// ---- VISUs/Manual_Camera_RawData.TcVIS
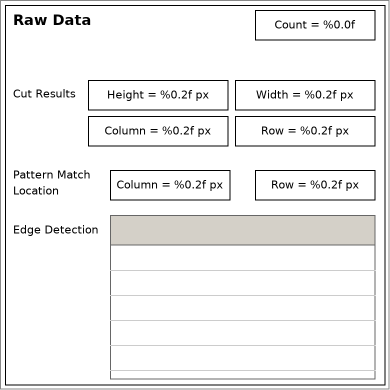
VISUALIZATION Manual_Camera_RawData  // 390x390
    Rectangle (5,5 380x380)
    Label (10,5 297x30), "Raw Data"
    Rectangle (255,10 120x30), "Count = %0.0f", text variable: MAIN.fbSlitter.Camera.CameraData.Results.Count
    Rectangle (110,170 120x30), "Column = %0.2f px", text variable: MAIN.fbSlitter.Camera.CameraData.Results.PatternMatchColumn
    Rectangle (255,170 120x30), "Row = %0.2f px", text variable: MAIN.fbSlitter.Camera.CameraData.Results.PatternMatchRow
    Rectangle (88,116 140x30), "Column = %0.2f px", text variable: MAIN.fbSlitter.Camera.CameraData.Results.LocationInX
    Rectangle (235,116 140x30), "Row = %0.2f px", text variable: MAIN.fbSlitter.Camera.CameraData.Results.LocationInY
    Rectangle (88,80 140x30), "Height = %0.2f px", text variable: MAIN.fbSlitter.Camera.CameraData.Results.HeightMeasurement
    Rectangle (235,80 140x30), "Width = %0.2f px", text variable: MAIN.fbSlitter.Camera.CameraData.Results.WidthMeasurement
    Label (10,215 101x30), "Edge Detection"
    Table (110,215 265x164), data array: MAIN.fbSlitter.Camera._displayVisionPts
        p1128707560: GVL.NumberVisionPoints
        p3854506369: MAIN.fbSlitter.Camera._displayVisionPts[1,INDEX]
        p1892666644: MAIN.fbSlitter.Camera._displayVisionPts[2,INDEX]
        p2232123230: Column
        p511219082: Row
    Group (10,160 96x46)
        Label (0,0 96x30), "Pattern Match"
        Label (0,16 96x30), "Location"
    Label (10,79 101x30), "Cut Results"
END_VISUALIZATION

// ---- VISUs/Manual_Cutter.TcVIS
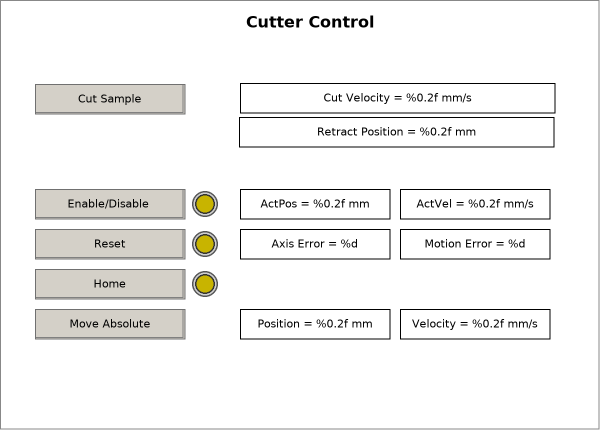
VISUALIZATION Manual_Cutter  // 600x430
    Label (133,7 355x30), "Cutter Control"
    Button (35,84 150x30), "Cut Sample", input disabled if: MAIN.fbSlitter.bBusy
        OnMouseClick: execute { MAIN.fbSlitter.Manual.bCutSample := TRUE; }
    Button (35,189 150x30), "Enable/Disable", input disabled if: MAIN.fbSlitter.bBusy
        OnMouseClick: execute { MAIN.fbSlitter.Manual.bCutterDisable := TRUE; }
    Button (35,229 150x30), "Reset", input disabled if: MAIN.fbSlitter.bBusy
        OnMouseClick: execute { MAIN.fbSlitter.Manual.bCutterReset := TRUE; }
    Button (35,269 150x30), "Home"
        OnMouseClick: execute { MAIN.fbSlitter.Manual.bCutterHome := TRUE; }
    Lamp1 (190,189 30x30), variable: MAIN.fbSlitter.Cutter.Axis.NcToPlc.StateDWord.0 = 1, style: Lamp-Lamp1-Yellow
    Rectangle (240,229 150x30), "Axis Error = %d", text variable: MAIN.fbSlitter.Cutter.Axis.NcToPlc.ErrorCode
    Lamp1 (190,229 30x30), variable: MAIN.fbSlitter.Cutter.Axis.NcToPlc.ErrorCode <> 0, style: Lamp-Lamp1-Yellow
    Lamp1 (190,269 30x30), variable: MAIN.fbSlitter.Cutter.Axis.NcToPlc.StateDWord.1 = 1, style: Lamp-Lamp1-Yellow
    Rectangle (400,229 150x30), "Motion Error = %d", text variable: MAIN.fbSlitter.Cutter._errorCode
    Button (35,309 150x30), "Move Absolute"
        OnMouseClick: execute { MAIN.fbSlitter.Manual.bCutterMoveAbs := TRUE; }
    Rectangle (240,309 150x30), "Position = %0.2f mm", text variable: MAIN.fbSlitter.Cutter._position
        OnMouseClick: write MAIN.fbSlitter.Cutter._position via Default, min 0, max 20, title 'Cutter Position'
    Rectangle (400,309 150x30), "Velocity = %0.2f mm/s", text variable: MAIN.fbSlitter.Cutter._velocity
        OnMouseClick: write MAIN.fbSlitter.Cutter._velocity via Default, title 'Cutter Velocity'
    Rectangle (240,189 150x30), "ActPos = %0.2f mm", text variable: MAIN.fbSlitter.Cutter.Axis.NcToPlc.ActPos
    Rectangle (400,189 150x30), "ActVel = %0.2f mm/s", text variable: MAIN.fbSlitter.Cutter.Axis.NcToPlc.ActVelo
    Rectangle (240,83 315x30), "Cut Velocity = %0.2f mm/s", text variable: MAIN.fbSlitter.Cutter._hmiParameters.cutVelocity
        OnMouseClick: write MAIN.fbSlitter.Cutter._hmiParameters.cutVelocity via Default, title 'Cutter Velocity'
    Rectangle (239,117 315x30), "Retract Position = %0.2f mm", text variable: MAIN.fbSlitter.Cutter._hmiParameters.retractPosition
        OnMouseClick: write MAIN.fbSlitter.Cutter._hmiParameters.retractPosition via Default, title 'Retract Position'
END_VISUALIZATION

// ---- VISUs/Manual_Ejector.TcVIS
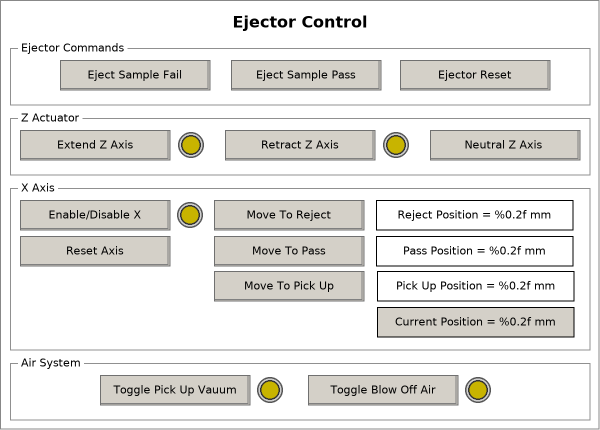
VISUALIZATION Manual_Ejector  // 600x430
    GroupBox (10,355 580x65), "Air System"
    Label (0,7 600x30), "Ejector Control"
    Button (100,375 150x30), "Toggle Pick Up Vauum"
        OnMouseClick: execute { MAIN.fbSlitter.Manual.bEjectVacuum := TRUE; }
    Button (308,375 150x30), "Toggle Blow Off Air"
        OnMouseClick: execute { MAIN.fbSlitter.Manual.bEjectBlowOff := TRUE; }
    Lamp1 (463,375 30x30), variable: MAIN.fbSlitter.Ejector._BlowOff, style: Lamp-Lamp1-Yellow
    Lamp1 (255,375 30x30), variable: MAIN.fbSlitter.Ejector._Vacuum, style: Lamp-Lamp1-Yellow
    Group (10,110 580x65)
        GroupBox (0,0 580x65), "Z Actuator"
        Button (10,20 150x30), "Extend Z Axis", input disabled if: MAIN.fbSlitter.bBusy
            OnMouseClick: execute { MAIN.fbSlitter.Manual.bEjectZExtend := TRUE; }
        Button (215,20 150x30), "Retract Z Axis", input disabled if: MAIN.fbSlitter.bBusy
            OnMouseClick: execute { MAIN.fbSlitter.Manual.bEjectZRetract := TRUE; }
        Button (420,20 150x30), "Neutral Z Axis", input disabled if: MAIN.fbSlitter.bBusy
            tap MAIN.fbSlitter.Manual.bEjectZOff
            OnMouseClick: execute { MAIN.fbSlitter.Manual.bEjectZNeutral := TRUE; }
        Lamp1 (166,20 30x30), variable: MAIN.fbSlitter.Ejector.zSlide.diExtended, style: Lamp-Lamp1-Yellow
        Lamp1 (371,20 30x30), variable: MAIN.fbSlitter.Ejector.zSlide.diRetracted, style: Lamp-Lamp1-Yellow
    GroupBox (10,40 580x65), "Ejector Commands"
        Button (390,20 150x30), "Ejector Reset", input disabled if: MAIN.fbSlitter.bBusy
            OnMouseClick: execute { MAIN.fbSlitter.Manual.bEjectReset := TRUE; }
    Button (60,60 150x30), "Eject Sample Fail", input disabled if: MAIN.fbSlitter.bBusy
        OnMouseClick: execute { MAIN.fbSlitter.Manual.bEjectSampleFail := TRUE; }
    Button (231,60 150x30), "Eject Sample Pass", input disabled if: MAIN.fbSlitter.bBusy
        OnMouseClick: execute { MAIN.fbSlitter.Manual.bEjectSamplePass := TRUE; }
    GroupBox (10,180 580x170), "X Axis"
        Rectangle (367,91 197x30), "Pick Up Position = %0.2f mm", text variable: MAIN.fbSlitter.Ejector._hmiParameters.ejectPositionHome
            OnMouseClick: write MAIN.fbSlitter.Ejector._hmiParameters.ejectPositionHome via Default, title 'Pick Up Position'
        Rectangle (367,127 197x30), "Current Position = %0.2f mm", text variable: MAIN.fbSlitter.Ejector.axis.axis.NcToPlc.ActPos
        Button (10,56 150x30), "Reset Axis"
            OnMouseClick: execute { MAIN.fbSlitter.Manual.bEjectAxisReset := TRUE; }
    Button (20,200 150x30), "Enable/Disable X", input disabled if: MAIN.fbSlitter.bBusy
        OnMouseClick: execute { MAIN.fbSlitter.Manual.bEjectAxisEnableToggle := TRUE; }
    Lamp1 (175,200 30x30), variable: MAIN.fbSlitter.Ejector.axis.axis.NcToPlc.StateDWord.0 = 1, style: Lamp-Lamp1-Yellow
    Button (214,200 150x30), "Move To Reject", input disabled if: MAIN.fbSlitter.bBusy
        OnMouseClick: execute { Main.fbSlitter.Manual.bEjectAxisFailPosition := TRUE; }
    Button (214,236 150x30), "Move To Pass", input disabled if: MAIN.fbSlitter.bBusy
        OnMouseClick: execute { Main.fbSlitter.Manual.bEjectAxisPassPosition := TRUE; }
    Button (214,271 150x30), "Move To Pick Up", input disabled if: MAIN.fbSlitter.bBusy
        OnMouseClick: execute { Main.fbSlitter.Manual.bEjectAxisHomePosition := TRUE; }
    Rectangle (376,200 197x30), "Reject Position = %0.2f mm", text variable: MAIN.fbSlitter.Ejector._hmiParameters.ejectPositionFail
        OnMouseClick: write MAIN.fbSlitter.Ejector._hmiParameters.ejectPositionFail via Default, title 'Reject Position'
    Rectangle (376,236 197x30), "Pass Position = %0.2f mm", text variable: MAIN.fbSlitter.Ejector._hmiParameters.ejectPositionPass
        OnMouseClick: write MAIN.fbSlitter.Ejector._hmiParameters.ejectPositionPass via Default, title 'Pass Position'
END_VISUALIZATION

// ---- VISUs/Manual_Frame.TcVIS
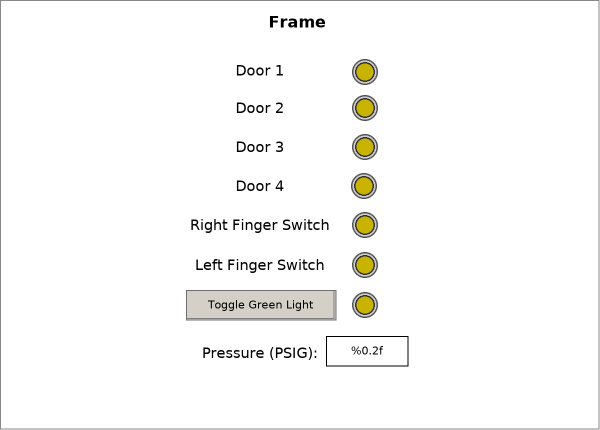
VISUALIZATION Manual_Frame  // 600x430
    Label (0,7 600x30), "Frame"
    Label (185,57 150x27), "Door 1"
    Label (185,93 150x30), "Door 2"
    Label (185,132 150x30), "Door 3"
    Label (185,210 150x30), "Right Finger Switch"
    Label (185,250 150x30), "Left Finger Switch"
    Lamp1 (350,57 30x30), variable: MAIN.Frame.diDoor1, style: Lamp-Lamp1-Yellow
    Lamp1 (350,93 30x30), variable: MAIN.Frame.diDoor2, style: Lamp-Lamp1-Yellow
    Lamp1 (350,132 30x30), variable: MAIN.Frame.diDoor3, style: Lamp-Lamp1-Yellow
    Lamp1 (350,210 30x30), variable: MAIN.Frame.diControlLeft, style: Lamp-Lamp1-Yellow
    Lamp1 (350,250 30x30), variable: MAIN.Frame.diControlRight, style: Lamp-Lamp1-Yellow
    Lamp1 (350,290 30x30), variable: MAIN.Frame.doGreen, style: Lamp-Lamp1-Yellow
    Button (186,290 150x30), "Toggle Green Light"
        OnMouseClick: execute { MAIN.Frame.GreenLight := NOT MAIN.Frame.GreenLight; }
    Label (185,338 150x30), "Pressure (PSIG):"
    Rectangle (326,336 82x30), "%0.2f", text variable: MAIN.Frame._pressure
    Label (185,171 150x30), "Door 4"
    Lamp1 (349,171 30x30), variable: MAIN.Frame.diDoor4, style: Lamp-Lamp1-Yellow
END_VISUALIZATION

// ---- VISUs/Manual_Mandrel.TcVIS
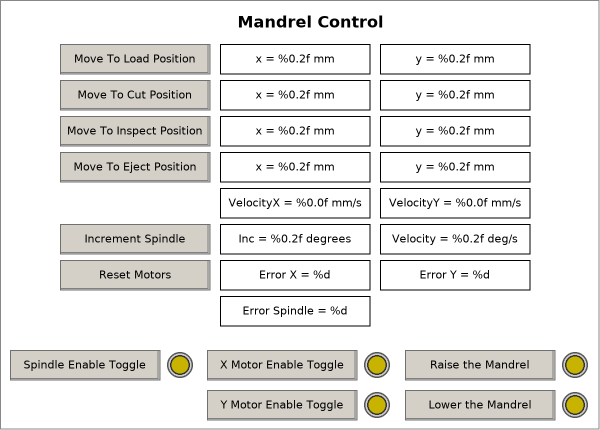
VISUALIZATION Manual_Mandrel  // 600x430
    Button (60,44 150x30), "Move To Load Position", input disabled if: MAIN.fbSlitter.bBusy
        OnMouseClick: execute { MAIN.fbSlitter.Manual.bMoveToLoadPosition := TRUE; }
    Button (60,80 150x30), "Move To Cut Position", input disabled if: MAIN.fbSlitter.bBusy
        OnMouseClick: execute { MAIN.fbSlitter.Manual.bMoveToCutPosition := TRUE; }
    Button (60,116 150x30), "Move To Inspect Position", input disabled if: MAIN.fbSlitter.bBusy
        OnMouseClick: execute { MAIN.fbSlitter.Manual.bMoveToInspectPosition := TRUE; }
    Button (60,152 150x30), "Move To Eject Position", input disabled if: MAIN.fbSlitter.bBusy
        OnMouseClick: execute { MAIN.fbSlitter.Manual.bMoveToEjectPosition := TRUE; }
    Button (405,350 150x30), "Raise the Mandrel", input disabled if: MAIN.fbSlitter.bBusy
        OnMouseClick: execute { MAIN.fbSlitter.Manual.bRaiseMandrel := TRUE; }
    Button (405,390 150x30), "Lower the Mandrel", input disabled if: MAIN.fbSlitter.bBusy
        OnMouseClick: execute { MAIN.fbSlitter.Manual.bLowerMandrel := TRUE; }
    Rectangle (220,44 150x30), "x = %0.2f mm", text variable: MAIN.fbSlitter.Mandrel._hmiParameters.loadPositionX
        OnMouseClick: write MAIN.fbSlitter.Mandrel._hmiParameters.loadPositionX via Default, title 'Load Position X'
    Rectangle (380,44 150x30), "y = %0.2f mm", text variable: MAIN.fbSlitter.Mandrel._hmiParameters.loadPositionY
        OnMouseClick: write MAIN.fbSlitter.Mandrel._hmiParameters.loadPositionY via Default, title 'Load Position Y'
    Rectangle (220,80 150x30), "x = %0.2f mm", text variable: MAIN.TubeHmi.CutPositionX
        OnMouseClick: write MAIN.TubeHmi.CutPositionX via Default, title 'Cut Position X'
    Rectangle (380,80 150x30), "y = %0.2f mm", text variable: MAIN.TubeHmi.CutPositionY
        OnMouseClick: write MAIN.TubeHmi.CutPositionY via Default, title 'Cut Position Y'
    Rectangle (220,116 150x30), "x = %0.2f mm", text variable: MAIN.TubeHmi.InspectPositionX
        OnMouseClick: write MAIN.TubeHmi.InspectPositionX via Default, title 'Inspect Position X'
    Rectangle (380,116 150x30), "y = %0.2f mm", text variable: MAIN.TubeHmi.InspectPositionY
        OnMouseClick: write MAIN.TubeHmi.InspectPositionY via Default, title 'Inspect Position Y'
    Rectangle (220,152 150x30), "x = %0.2f mm", text variable: MAIN.TubeHmi.EjectPositionX
        OnMouseClick: write MAIN.TubeHmi.EjectPositionX via Default, title 'Eject Position X'
    Rectangle (380,152 150x30), "y = %0.2f mm", text variable: MAIN.TubeHmi.EjectPositionY
        OnMouseClick: write MAIN.TubeHmi.EjectPositionY via Default, title 'Eject Position Y'
    Lamp1 (560,350 30x30), variable: MAIN.fbSlitter.Mandrel.doStripperExtend AND NOT MAIN.fbSlitter.Mandrel.doStripperRetract, style: Lamp-Lamp1-Yellow
    Lamp1 (560,390 30x30), variable: NOT MAIN.fbSlitter.Mandrel.doStripperExtend AND MAIN.fbSlitter.Mandrel.doStripperRetract, style: Lamp-Lamp1-Yellow
    Rectangle (220,188 150x30), "VelocityX = %0.0f mm/s", text variable: MAIN.fbSlitter.Mandrel._hmiParameters.velocityX
        OnMouseClick: write MAIN.fbSlitter.Mandrel._hmiParameters.velocityX via Default, title 'Velocity X'
    Rectangle (380,188 150x30), "VelocityY = %0.0f mm/s", text variable: MAIN.fbSlitter.Mandrel._hmiParameters.velocityY
        OnMouseClick: write MAIN.fbSlitter.Mandrel._hmiParameters.velocityY via Default, title 'Velocity Y'
    Rectangle (220,260 150x30), "Error X = %d", text variable: MAIN.fbSlitter.Mandrel.Xaxis.NcToPlc.ErrorCode
    Rectangle (380,260 150x30), "Error Y = %d", text variable: MAIN.fbSlitter.Mandrel.Yaxis.NcToPlc.ErrorCode
    Button (60,260 150x30), "Reset Motors"
        OnMouseClick: execute { MAIN.fbSlitter.Manual.bMandrelReset := TRUE; }
    Button (207,350 150x30), "X Motor Enable Toggle", input disabled if: MAIN.fbSlitter.bBusy
        OnMouseClick: execute { MAIN.fbSlitter.Manual.bMandrelXEnableToggle := TRUE; }
    Button (207,390 150x30), "Y Motor Enable Toggle", input disabled if: MAIN.fbSlitter.bBusy
        OnMouseClick: execute { MAIN.fbSlitter.Manual.bMandrelYEnableToggle := TRUE; }
    Button (10,350 150x30), "Spindle Enable Toggle"
        OnMouseClick: execute { MAIN.fbSlitter.Manual.bMandrelSpindleToggle := TRUE; }
    Lamp1 (362,350 30x30), variable: MAIN.fbSlitter.Mandrel.Xaxis.NcToPlc.StateDWord.0 = 1, style: Lamp-Lamp1-Yellow
    Lamp1 (165,350 30x30), variable: MAIN.fbSlitter.Mandrel.Spindle.NcToPlc.StateDWord.0 = 1, style: Lamp-Lamp1-Yellow
    Lamp1 (362,390 30x30), variable: MAIN.fbSlitter.Mandrel.Yaxis.NcToPlc.StateDWord.0 = 1, style: Lamp-Lamp1-Yellow
    Label (133,7 355x30), "Mandrel Control"
    Rectangle (220,296 150x30), "Error Spindle = %d", text variable: MAIN.fbSlitter.Mandrel.Spindle.NcToPlc.ErrorCode
    Button (60,224 150x30), "Increment Spindle", input disabled if: MAIN.fbSlitter.bBusy
        OnMouseClick: execute { MAIN.fbSlitter.Manual.bMandrelSpindleRotate := TRUE; }
    Rectangle (220,224 150x30), "Inc = %0.2f degrees", text variable: MAIN.fbSlitter.Mandrel._SpindleIncrement
        OnMouseClick: write MAIN.fbSlitter.Mandrel._SpindleIncrement via Default, title 'Spingle Increment'
    Rectangle (380,224 150x30), "Velocity = %0.2f deg/s", text variable: MAIN.fbSlitter.Mandrel._hmiParameters.spindleVelocity
        OnMouseClick: write MAIN.fbSlitter.Mandrel._hmiParameters.spindleVelocity via Default, title 'Spindle Velocity'
END_VISUALIZATION

// ---- VISUs/Manual_Vacuum.TcVIS
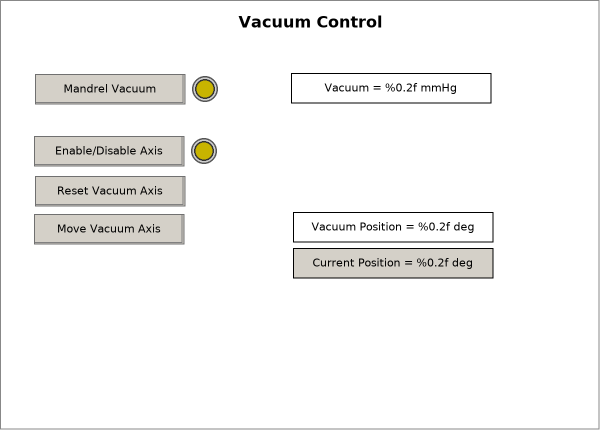
VISUALIZATION Manual_Vacuum  // 600x430
    Label (133,7 355x30), "Vacuum Control"
    Rectangle (291,73 200x30), "Vacuum = %0.2f mmHg", text variable: MAIN.fbSlitter.Mandrel._vacuum_mmHg
    Button (35,74 150x30), "Mandrel Vacuum"
        OnMouseClick: execute { MAIN.fbSlitter.Manual.bToggleMandrelVacuum := TRUE; }
    Lamp1 (190,74 30x30), variable: MAIN.fbSlitter.Mandrel.doVacuum, style: Lamp-Lamp1-Yellow
    Button (34,136 150x30), "Enable/Disable Axis"
        OnMouseClick: execute { MAIN.fbSlitter.Manual.bVacuumAxisToggleEnable := TRUE; }
    Lamp1 (189,136 30x30), variable: MAIN.fbSlitter.Mandrel.VacAxis.axis.NcToPlc.StateDWord.0 = 1, style: Lamp-Lamp1-Yellow
    Rectangle (293,248 200x30), "Current Position = %0.2f deg", text variable: MAIN.fbSlitter.Mandrel.VacAxis.axis.NcToPlc.ActPos
    Rectangle (293,212 200x30), "Vacuum Position = %0.2f deg", text variable: MAIN.TubeHmi.VacPosition
        OnMouseClick: write MAIN.TubeHmi.VacPosition via Default, min 0, max 13000, title 'Vacuum Position'
    Button (34,214 150x30), "Move Vacuum Axis"
        OnMouseClick: execute { MAIN.fbSlitter.Manual.bVacuumAxisMove := TRUE; }
    Button (35,176 150x30), "Reset Vacuum Axis"
        OnMouseClick: execute { MAIN.fbSlitter.Manual.bVacuumAxisReset := TRUE; }
END_VISUALIZATION

// ---- VISUs/Manual_Select_Tube.TcVIS
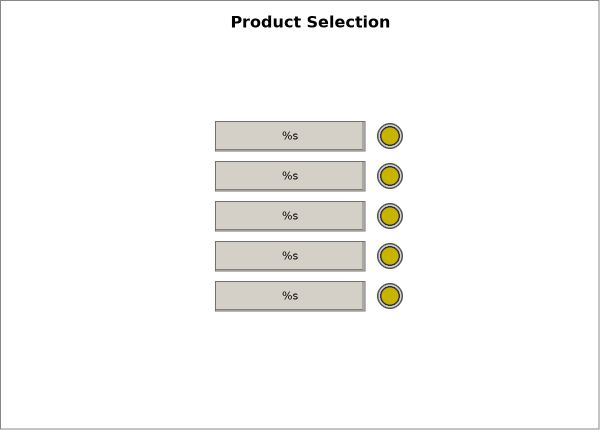
VISUALIZATION Manual_Select_Tube  // 600x430
    Button (215,121 150x30), "%s", text variable: MAIN.TubeSelection[1].ProductName
        OnMouseClick: execute {
            MAIN.TubeHmi := MAIN.TubeSelection[1];
            MAIN.fbSlitter.Manual.bCameraSelectTube := TRUE;
            MAIN.TubeIndicator[1] := TRUE;
            MAIN.TubeIndicator[2] := FALSE;
            MAIN.TubeIndicator[3] := FALSE;
            MAIN.TubeIndicator[4] := FALSE;
            MAIN.TubeIndicator[5] := FALSE;
        }
    Button (215,161 150x30), "%s", text variable: MAIN.TubeSelection[2].ProductName
        OnMouseClick: execute {
            MAIN.TubeHmi := MAIN.TubeSelection[2];
            MAIN.fbSlitter.Manual.bCameraSelectTube := TRUE;
            MAIN.TubeIndicator[1] := FALSE;
            MAIN.TubeIndicator[2] := TRUE;
            MAIN.TubeIndicator[3] := FALSE;
            MAIN.TubeIndicator[4] := FALSE;
            MAIN.TubeIndicator[5] := FALSE;
        }
    Button (215,201 150x30), "%s", text variable: MAIN.TubeSelection[3].ProductName
        OnMouseClick: execute {
            MAIN.TubeHmi := MAIN.TubeSelection[3];
            MAIN.fbSlitter.Manual.bCameraSelectTube := TRUE;
            MAIN.TubeIndicator[1] := FALSE;
            MAIN.TubeIndicator[2] := FALSE;
            MAIN.TubeIndicator[3] := TRUE;
            MAIN.TubeIndicator[4] := FALSE;
            MAIN.TubeIndicator[5] := FALSE;
        }
    Button (215,241 150x30), "%s", text variable: MAIN.TubeSelection[4].ProductName
        OnMouseClick: execute {
            MAIN.TubeHmi := MAIN.TubeSelection[4];
            MAIN.fbSlitter.Manual.bCameraSelectTube := TRUE;
            MAIN.TubeIndicator[1] := FALSE;
            MAIN.TubeIndicator[2] := FALSE;
            MAIN.TubeIndicator[3] := FALSE;
            MAIN.TubeIndicator[4] := TRUE;
            MAIN.TubeIndicator[5] := FALSE;
        }
    Button (215,281 150x30), "%s", text variable: MAIN.TubeSelection[5].ProductName
        OnMouseClick: execute {
            MAIN.TubeHmi := MAIN.TubeSelection[5];
            MAIN.fbSlitter.Manual.bCameraSelectTube := TRUE;
            MAIN.TubeIndicator[1] := FALSE;
            MAIN.TubeIndicator[2] := FALSE;
            MAIN.TubeIndicator[3] := FALSE;
            MAIN.TubeIndicator[4] := FALSE;
            MAIN.TubeIndicator[5] := TRUE;
        }
    Lamp1 (375,121 30x30), variable: MAIN.TubeIndicator[1], style: Lamp-Lamp1-Yellow
    Lamp1 (375,161 30x30), variable: MAIN.TubeIndicator[2], style: Lamp-Lamp1-Yellow
    Lamp1 (375,201 30x30), variable: MAIN.TubeIndicator[3], style: Lamp-Lamp1-Yellow
    Lamp1 (375,241 30x30), variable: MAIN.TubeIndicator[4], style: Lamp-Lamp1-Yellow
    Lamp1 (375,281 30x30), variable: MAIN.TubeIndicator[5], style: Lamp-Lamp1-Yellow
    Label (133,7 355x30), "Product Selection"
END_VISUALIZATION

// ---- VISUs/Settings.TcVIS
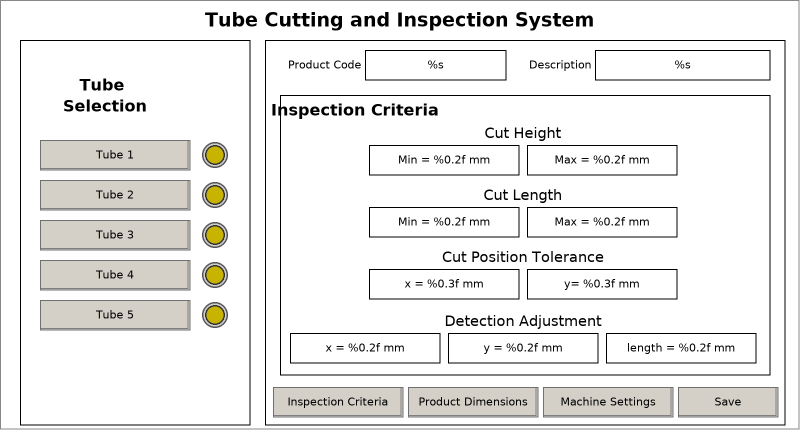
VISUALIZATION Settings  // 800x430
    Frame (255,30 540x400)
        shows SettingsTemplate(Tube := MAIN.TubeHmi)
        shows SettingsTemplate(Tube := MAIN.TubeSelection[2])
        shows SettingsTemplate(Tube := MAIN.TubeSelection[3])
        shows SettingsTemplate(Tube := MAIN.TubeSelection[4])
        shows SettingsTemplate(Tube := MAIN.TubeSelection[5])
    Label (10,79 170x30)
    Label (0,5 800x30), "Tube Cutting and Inspection System"
    Group (20,65 230x51)
        Label (0,21 170x30), "Selection"
        Label (0,0 170x30), "Tube"
    Rectangle (20,40 230x385)
    Button (40,140 150x30), "Tube 1"
        OnMouseClick: execute {
            MAIN.TubeHmi := MAIN.TubeSelection[1];
            MAIN.TubeIndicator[1] := TRUE;
            MAIN.TubeIndicator[2] := FALSE;
            MAIN.TubeIndicator[3] := FALSE;
            MAIN.TubeIndicator[4] := FALSE;
            MAIN.TubeIndicator[5] := FALSE;
        }
    Button (40,180 150x30), "Tube 2"
        OnMouseClick: execute {
            MAIN.TubeHmi := MAIN.TubeSelection[2];
            MAIN.TubeIndicator[1] := FALSE;
            MAIN.TubeIndicator[2] := TRUE;
            MAIN.TubeIndicator[3] := FALSE;
            MAIN.TubeIndicator[4] := FALSE;
            MAIN.TubeIndicator[5] := FALSE;
        }
    Button (40,220 150x30), "Tube 3"
        OnMouseClick: execute {
            MAIN.TubeHmi := MAIN.TubeSelection[3];
            MAIN.TubeIndicator[1] := FALSE;
            MAIN.TubeIndicator[2] := FALSE;
            MAIN.TubeIndicator[3] := TRUE;
            MAIN.TubeIndicator[4] := FALSE;
            MAIN.TubeIndicator[5] := FALSE;
        }
    Button (40,260 150x30), "Tube 4"
        OnMouseClick: execute {
            Main.TubeHmi := MAIN.TubeSelection[4];
            MAIN.TubeIndicator[1] := FALSE;
            MAIN.TubeIndicator[2] := FALSE;
            MAIN.TubeIndicator[3] := FALSE;
            MAIN.TubeIndicator[4] := TRUE;
            MAIN.TubeIndicator[5] := FALSE;
        }
    Button (40,300 150x30), "Tube 5"
        OnMouseClick: execute {
            Main.TubeHmi := MAIN.TubeSelection[5];
            MAIN.TubeIndicator[1] := FALSE;
            MAIN.TubeIndicator[2] := FALSE;
            MAIN.TubeIndicator[3] := FALSE;
            MAIN.TubeIndicator[4] := FALSE;
            MAIN.TubeIndicator[5] := TRUE;
        }
    Lamp1 (200,140 30x30), variable: MAIN.TubeIndicator[1], style: Lamp-Lamp1-Yellow
    Lamp1 (200,180 30x30), variable: MAIN.TubeIndicator[2], style: Lamp-Lamp1-Yellow
    Lamp1 (200,220 30x30), variable: MAIN.TubeIndicator[3], style: Lamp-Lamp1-Yellow
    Lamp1 (200,260 30x30), variable: MAIN.TubeIndicator[4], style: Lamp-Lamp1-Yellow
    Lamp1 (200,300 30x30), variable: MAIN.TubeIndicator[5], style: Lamp-Lamp1-Yellow
    Group (20,70 230x51)
        Label (0,21 170x30), "Selection"
        Label (0,0 170x30), "Tube"
END_VISUALIZATION

// ---- VISUs/SettingsTemplate.TcVIS
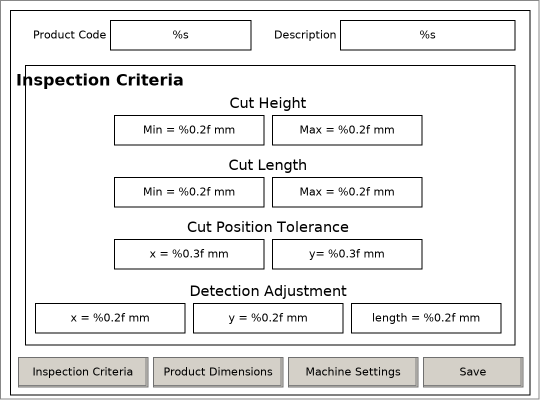
VISUALIZATION SettingsTemplate  // 540x400
VAR_IN_OUT
	Tube : ST_TubeParameters;
END_VAR
    Rectangle (10,10 520x385)
    Rectangle (110,20 141x30), "%s", text variable: Tube.ProductName
        OnMouseClick: write Tube.ProductName via Default
    Label (30,20 80x30), "Product Code"
    Button (288,357 130x30), "Machine Settings"
        OnMouseClick: FrameSelectionChange Selection=SelectedFrame=c09837a4-7cd0-42f3-a923-2461df8b3e92, Selection=1, GlobSel=AssignType=Directly, SelType=Locally
    Button (18,357 130x30), "Inspection Criteria"
        OnMouseClick: FrameSelectionChange Selection=SelectedFrame=c09837a4-7cd0-42f3-a923-2461df8b3e92, GlobSel=AssignType=Directly, SelType=Locally
    Button (153,357 130x30), "Product Dimensions"
        OnMouseClick: FrameSelectionChange Selection=SelectedFrame=c09837a4-7cd0-42f3-a923-2461df8b3e92, Selection=2, GlobSel=AssignType=Directly, SelType=Locally
    Button (423,357 100x30), "Save"
        OnMouseClick: execute { MAIN.bSave := TRUE; }
    Frame (15,55 510x300)
        shows Settings_PassCriteria(CutHeightMin := Tube.MinHeight, CutHeightMax := Tube.MaxHeight, CutLengthMin := Tube.MinLength, CutLengthMax := Tube.MaxLength, CutToleranceX := Tube.ResultToleranceX, CutToleranceY := Tube.ResultToleranceY, AdjustmentX := Tube.AdjustmentX, AdjustmentY := Tube.AdjustmentY, AdjustmentLength := Tube.AdjustmentLength)
        shows Settings_Mandrel(CutPositionX := Tube.CutPositionX, CutPositionY := Tube.CutPositionY, InspectPositionX := Tube.InspectPositionX, InspectPositionY := Tube.InspectPositionY, EjectPositionX := Tube.EjectPositionX, EjectPositionY := Tube.EjectPositionY, VacuumThreshold := Tube.VacuumThreshold, VacuumPosition := Tube.VacPosition)
        shows Settings_ProductDimensions(Diameter := Tube.Diameter, PocketDepth := Tube.DepthOfPocket)
    Label (271,20 69x30), "Description"
    Rectangle (340,20 175x30), "%s", text variable: Tube.Description
        OnMouseClick: write Tube.Description via Default
END_VISUALIZATION

// ---- VISUs/Settings_Mandrel.TcVIS
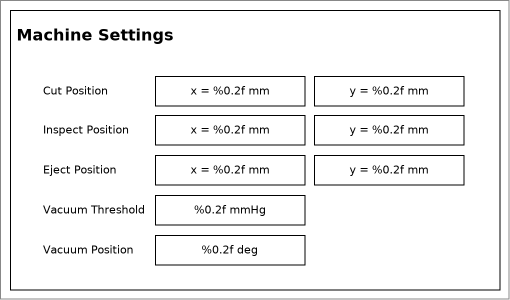
VISUALIZATION Settings_Mandrel  // 510x300
VAR_IN_OUT
	CutPositionX	: LREAL;
	CutPositionY	: LREAL;
	InspectPositionX: LREAL;
	InspectPositionY: LREAL;
	EjectPositionX	: LREAL;
	EjectPositionY	: LREAL;
	VacuumThreshold	: REAL;
	VacuumPosition : LREAL;
END_VAR
    Rectangle (10,10 490x280)
    Label (20,20 150x30), "Machine Settings"
    Label (40,76 90x30), "Cut Position"
    Label (40,115 90x30), "Inspect Position"
    Label (40,155 90x30), "Eject Position"
    Rectangle (155,76 150x30), "x = %0.2f mm", text variable: CutPositionX
        OnMouseClick: write CutPositionX via Default
    Rectangle (314,76 150x30), "y = %0.2f mm", text variable: CutPositionY
        OnMouseClick: write CutPositionY via Default
    Rectangle (155,115 150x30), "x = %0.2f mm", text variable: InspectPositionX
        OnMouseClick: write InspectPositionX via Default
    Rectangle (314,115 150x30), "y = %0.2f mm", text variable: InspectPositionY
        OnMouseClick: write InspectPositionY via Default
    Rectangle (155,155 150x30), "x = %0.2f mm", text variable: EjectPositionX
        OnMouseClick: write EjectPositionX via Default
    Rectangle (314,155 150x30), "y = %0.2f mm", text variable: EjectPositionY
        OnMouseClick: write EjectPositionY via Default
    Label (40,195 110x30), "Vacuum Threshold"
    Rectangle (155,195 150x30), "%0.2f mmHg", text variable: VacuumThreshold
        OnMouseClick: write VacuumThreshold via Default
    Label (40,235 110x30), "Vacuum Position"
    Rectangle (155,235 150x30), "%0.2f deg", text variable: VacuumPosition
        OnMouseClick: write VacuumPosition via Default, min 0, max 13000, title 'Vacuum Axis Position'
END_VISUALIZATION

// ---- VISUs/Settings_PassCriteria.TcVIS
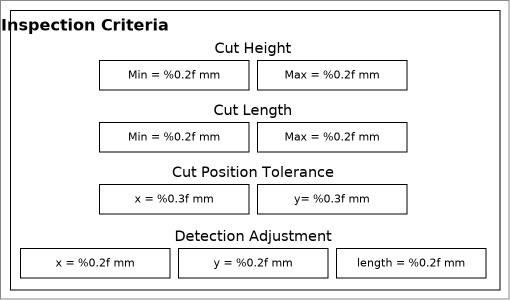
VISUALIZATION Settings_PassCriteria  // 510x300
VAR_IN_OUT
	CutHeightMin	: LREAL;
	CutHeightMax	: LREAL;
	CutLengthMin	: LREAL;
	CutLengthMax	: LREAL;
	CutToleranceX	: LREAL;
	CutToleranceY	: LREAL;
	AdjustmentX		: LREAL;
	AdjustmentY		: LREAL;
	AdjustmentLength: LREAL;
END_VAR
    Rectangle (10,10 490x280)
    Label (203,95 100x30), "Cut Length"
    Rectangle (99,122 150x30), "Min = %0.2f mm", text variable: CutLengthMin
        OnMouseClick: write CutLengthMin via Default
    Rectangle (257,122 150x30), "Max = %0.2f mm", text variable: CutLengthMax
        OnMouseClick: write CutLengthMax via Default, title 'Cut Position Y'
    Label (213,33 80x30), "Cut Height"
    Rectangle (99,60 150x30), "Min = %0.2f mm", text variable: CutHeightMin
        OnMouseClick: write CutHeightMin via Default
    Rectangle (257,60 150x30), "Max = %0.2f mm", text variable: CutHeightMax
        OnMouseClick: write CutHeightMax via Default, title 'Cut Position Y'
    Label (168,157 170x30), "Cut Position Tolerance"
    Rectangle (99,184 150x30), "x = %0.3f mm", text variable: CutToleranceX
        OnMouseClick: write CutToleranceX via Default
    Rectangle (257,184 150x30), "y= %0.3f mm", text variable: CutToleranceY
        OnMouseClick: write CutToleranceY via Default, title 'Cut Position Y'
    Label (173,221 160x30), "Detection Adjustment"
    Rectangle (20,248 150x30), "x = %0.2f mm", text variable: AdjustmentX
        OnMouseClick: write AdjustmentX via Default, title 'Cut Position X'
    Rectangle (178,248 150x30), "y = %0.2f mm", text variable: AdjustmentY
        OnMouseClick: write AdjustmentY via Default, title 'Cut Position Y'
    Rectangle (336,248 150x30), "length = %0.2f mm", text variable: AdjustmentLength
        OnMouseClick: write AdjustmentLength via Default, title 'Cut Position Y'
    Label (10,10 150x30), "Inspection Criteria"
END_VISUALIZATION

// ---- VISUs/Settings_ProductDimensions.TcVIS
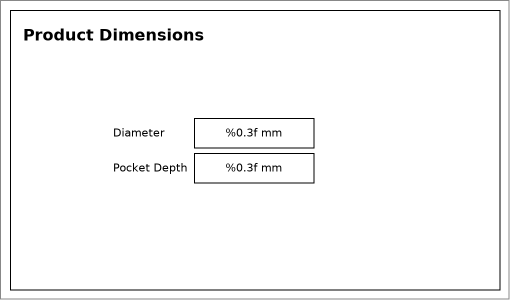
VISUALIZATION Settings_ProductDimensions  // 510x300
VAR_IN_OUT
	Diameter	: LREAL;
	PocketDepth	: LREAL;
END_VAR
    Rectangle (10,10 490x280)
    Group (110,118 204x65)
        Label (0,0 60x30), "Diameter"
        Rectangle (84,0 120x30), "%0.3f mm", text variable: Diameter
            OnMouseClick: write Diameter via Default
        Rectangle (84,35 120x30), "%0.3f mm", text variable: PocketDepth
            OnMouseClick: write PocketDepth via Default
        Label (0,35 80x30), "Pocket Depth"
    Label (20,20 150x30), "Product Dimensions"
END_VISUALIZATION

// ---- VISUs/Visualization.TcVIS
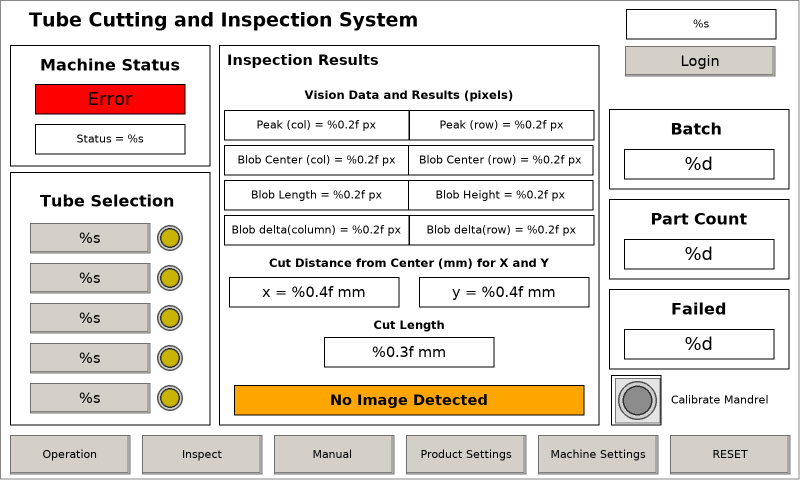
VISUALIZATION Visualization  // 800x480
    Button (10,435 120x39), "Operation"
        OnMouseClick: FrameSelectionChange Selection=SelectedFrame=9a7dff5b-3db9-4aa8-8ed3-29e44fa354e5, GlobSel=AssignType=Directly, SelType=Locally
        OnMouseClick: execute {
            MAIN.eModeCommand := E_PMLProtectedUnitMode.ePMLProtUnitMode_Production;
            MAIN.bOperation := TRUE;
            MAIN.bInspect := FALSE;
        }
    Button (274,435 120x39), "Manual"
        OnMouseClick: FrameSelectionChange Selection=SelectedFrame=9a7dff5b-3db9-4aa8-8ed3-29e44fa354e5, Selection=1, GlobSel=AssignType=Directly, SelType=Locally
        OnMouseClick: execute { Main.eModeCommand := E_PMLProtectedUnitMode.ePMLProtUnitMode_Manual; Main.bManual := TRUE; }
    Button (538,435 120x39), "Machine Settings"
        OnMouseClick: FrameSelectionChange Selection=SelectedFrame=9a7dff5b-3db9-4aa8-8ed3-29e44fa354e5, Selection=3, GlobSel=AssignType=Directly, SelType=Locally
        OnMouseClick: execute { MAIN.bMachineSettings := TRUE; }
    Frame (0,0 800x430)
        shows Front_Panel()
        shows ManualControl()
        shows Settings()
        shows MachineSettings()
        shows Manual_Inspect()
    Button (670,435 120x39), "RESET"
        OnMouseClick: execute { MAIN.hmiReset := TRUE; }
    Button (406,435 120x39), "Product Settings"
        OnMouseClick: FrameSelectionChange Selection=SelectedFrame=9a7dff5b-3db9-4aa8-8ed3-29e44fa354e5, Selection=2, GlobSel=AssignType=Directly, SelType=Locally
        OnMouseClick: execute { MAIN.bProductSettings := TRUE; }
    Button (142,435 120x39), "Inspect"
        OnMouseClick: FrameSelectionChange Selection=SelectedFrame=9a7dff5b-3db9-4aa8-8ed3-29e44fa354e5, Selection=4, GlobSel=AssignType=Directly, SelType=Locally
        OnMouseClick: execute {
            MAIN.eModeCommand := E_PMLProtectedUnitMode.ePMLProtUnitMode_Production;
            MAIN.bOperation := TRUE;
            MAIN.bInspect := TRUE;
        }
END_VISUALIZATION
